// TwinCAT 3 PLC project PalettenstationPLC
// ProgramVersion: 3.1.4022.7
// libraries:
//   Tc2_Standard, * (Beckhoff Automation GmbH)
//   Tc2_System, * (Beckhoff Automation GmbH)
//   Tc3_Module, * (Beckhoff Automation GmbH)
// project tree:
//   GVLs/ GVL_IO.TcGVL, GVL_Simulation.TcGVL
//   / PlcTask.TcTTO
//   POUs/ MAIN.TcPOU, FB_NotHalt.TcPOU
//   DUTs/ E_StoppKategorie.TcDUT
// real-time tasks:
//   TASK PlcTask: cycle T#10ms, priority 20, ADS port 350
//   TASK Task_IO: cycle T#10ms, priority 1, ADS port 301
// I/O:
//   DEVICE Gerät 1 (EtherCAT), AmsNetId 5.35.203.54.2.1
//     Klemme 1 (EK1100) [EK1100 EtherCAT-Koppler (2A E-Bus)]
//       Klemme 2 (EL1002) [EL1002 2K. Dig. Eingang 24V, 3ms]
//       Klemme 3 (EL1004) [EL1004 4K. Dig. Eingang 24V, 3ms]
//       Klemme 4 (EL1004) [EL1004 4K. Dig. Eingang 24V, 3ms]
//       Klemme 5 (EL1008) [EL1008 8K. Dig. Eingang 24V, 3ms]
//       Klemme 6 (EL2004) [EL2004 4K. Dig. Ausgang 24V, 0.5A]
//       Klemme 7 (EL2004) [EL2004 4K. Dig. Ausgang 24V, 0.5A]
//       Klemme 8 (EL2008) [EL2008 8K. Dig. Ausgang 24V, 0.5A]
//       Klemme 9 (EL3064) [EL3064 4K.Ana. Eingang 0-10V]
//       Klemme 10 (EL3144) [EL3144 4K. Ana. Eingang 0-20mA]
//       Klemme 11 (EL3204) [EL3204 4K. Ana. Eingang PT100 (RTD)]
//       Klemme 12 (EL4014) [EL4014 4K. Ana. Ausgang 0-20mA, 12bit]
//       Klemme 13 (EL3681) [EL3681 Digitale Multimeter Klemme]
//       Klemme 14 (EK1110) [EK1110 EtherCAT-Verlängerung]

CONFIGURATION PalettenstationPLC
    RESOURCE PLC ON TwinCAT3
        TASK PlcTask(INTERVAL := T#10ms, PRIORITY := 20);
        PROGRAM MAIN WITH PlcTask : MAIN;
    END_RESOURCE
END_CONFIGURATION

// ---- DUTs/E_StoppKategorie.TcDUT
// =====================================================
// E_StoppKategorie
// =====================================================
// Bildet die Stoppkategorien nach EN 60204-1 als Software-Modell ab
// (siehe FB_NotHalt fuer den ausfuehrlichen Sicherheitshinweis).
// KEINE zertifizierte Sicherheitsklassifizierung.
// =====================================================
TYPE E_StoppKategorie :
(
	Kategorie_0 := 0,	// Sofortiger, unkontrollierter Halt durch Wegnahme der Energie/Freigabe
	Kategorie_1 := 1	// Kontrollierter Halt: Energie bleibt bis sicherer Zustand erhalten, danach Wegnahme
);
END_TYPE

// ---- GVLs/GVL_IO.TcGVL
{attribute 'qualified_only'}
VAR_GLOBAL

    // ==================================================
    // DIGITALE EINGÄNGE
    // ==================================================

    DI_NotHaltFrei        AT %I* : BOOL;
    DI_SchutzhaubeZu      AT %I* : BOOL;
    DI_PaletteEingang     AT %I* : BOOL;
    DI_PalettePositioniert AT %I* : BOOL;
    DI_HubUnten           AT %I* : BOOL;
    DI_HubOben            AT %I* : BOOL;
    DI_KollisionFrei      AT %I* : BOOL;
    DI_WerkerQuittierung  AT %I* : BOOL;


    // ==================================================
    // DIGITALE AUSGÄNGE
    // ==================================================

    DO_SignalGruen        AT %Q* : BOOL;
    DO_AlarmRot           AT %Q* : BOOL;
    DO_Foerderband        AT %Q* : BOOL;
    DO_FoerderbandStopp   AT %Q* : BOOL;
    DO_HubwerkHoch        AT %Q* : BOOL;
    DO_HubwerkRunter      AT %Q* : BOOL;
    DO_ProzessFreigabe    AT %Q* : BOOL;
    DO_Heizfreigabe       AT %Q* : BOOL;


    // ==================================================
    // ANALOGE EINGÄNGE
    // ==================================================

    AI_FolienTemperatur   AT %I* : REAL;
    AI_MotorTemperatur    AT %I* : REAL;

	// ==================================================
	// INTERNE PROGRAMMVARIABLEN
	// ==================================================

	Schritt : INT := 0;
	AlarmAktiv : BOOL := FALSE;

	// SIM_Aktiv = TRUE  -> Schrittkette nutzt GVL_Simulation-Werte
	// SIM_Aktiv = FALSE -> Schrittkette nutzt echte DI_*-Hardwareeingaenge (Default)
	SIM_Aktiv : BOOL := FALSE;


END_VAR

// ---- GVLs/GVL_Simulation.TcGVL
{attribute 'qualified_only'}
VAR_GLOBAL
	GVL_SIM_NotHaltFrei         : BOOL := TRUE;
    GVL_SIM_SchutzhaubeZu       : BOOL := TRUE;
    GVL_SIM_PaletteEingang      : BOOL := FALSE;
    GVL_SIM_PalettePositioniert : BOOL := FALSE;
    GVL_SIM_HubUnten            : BOOL := TRUE;
    GVL_SIM_HubOben             : BOOL := FALSE;
    GVL_SIM_KollisionFrei       : BOOL := TRUE;
    GVL_SIM_WerkerQuittierung   : BOOL := FALSE;
	GVL_SIM_FolienTemperatur  	: REAL := 175.0;
	GVL_SIM_MotorTemperatur   	: REAL := 50.0;
	
END_VAR

// ---- POUs/MAIN.TcPOU
PROGRAM MAIN
VAR
	tProzesszeit : TON;

	bNotHaltFrei         : BOOL;
    bSchutzhaubeZu       : BOOL;
    bPaletteEingang      : BOOL;
    bPalettePositioniert : BOOL;
    bHubUnten            : BOOL;
    bHubOben             : BOOL;
    bKollisionFrei       : BOOL;
    bWerkerQuittierung   : BOOL;

END_VAR

// =====================================================
// AUSGÄNGE ZU BEGINN JEDES SPS-ZYKLUS ZURÜCKSETZEN
// =====================================================

GVL_IO.DO_SignalGruen      := FALSE;
GVL_IO.DO_AlarmRot         := FALSE;
GVL_IO.DO_Foerderband      := FALSE;
GVL_IO.DO_FoerderbandStopp := FALSE;
GVL_IO.DO_HubwerkHoch      := FALSE;
GVL_IO.DO_HubwerkRunter    := FALSE;
GVL_IO.DO_ProzessFreigabe  := FALSE;
GVL_IO.DO_Heizfreigabe     := FALSE;


// =====================================================
// UMSCHALTUNG SIMULATION / HARDWARE
// =====================================================
// GVL_IO.SIM_Aktiv = TRUE  -> Werte aus GVL_Simulation
// GVL_IO.SIM_Aktiv = FALSE -> Werte von den echten %I*-Eingaengen (Default)

IF GVL_IO.SIM_Aktiv THEN

    bNotHaltFrei         := GVL_Simulation.GVL_SIM_NotHaltFrei;
    bSchutzhaubeZu       := GVL_Simulation.GVL_SIM_SchutzhaubeZu;
    bPaletteEingang      := GVL_Simulation.GVL_SIM_PaletteEingang;
    bPalettePositioniert := GVL_Simulation.GVL_SIM_PalettePositioniert;
    bHubUnten            := GVL_Simulation.GVL_SIM_HubUnten;
    bHubOben             := GVL_Simulation.GVL_SIM_HubOben;
    bKollisionFrei       := GVL_Simulation.GVL_SIM_KollisionFrei;
    bWerkerQuittierung   := GVL_Simulation.GVL_SIM_WerkerQuittierung;
	
    GVL_IO.AI_FolienTemperatur := GVL_Simulation.GVL_SIM_FolienTemperatur;
	GVL_IO.AI_MotorTemperatur  := GVL_Simulation.GVL_SIM_MotorTemperatur;
	
	

ELSE

    bNotHaltFrei         := GVL_IO.DI_NotHaltFrei;
    bSchutzhaubeZu       := GVL_IO.DI_SchutzhaubeZu;
    bPaletteEingang      := GVL_IO.DI_PaletteEingang;
    bPalettePositioniert := GVL_IO.DI_PalettePositioniert;
    bHubUnten            := GVL_IO.DI_HubUnten;
    bHubOben             := GVL_IO.DI_HubOben;
    bKollisionFrei       := GVL_IO.DI_KollisionFrei;
    bWerkerQuittierung   := GVL_IO.DI_WerkerQuittierung;

END_IF

// lesen -->  Programm ausführen -->  E/A schreiben --> wieder von vorne
// =====================================================
// SCHRITTKETTE
// =====================================================

CASE GVL_IO.Schritt OF

    0:// S0 - Anlage bereit und wartet auf Palette

        GVL_IO.DO_SignalGruen := TRUE;

        IF bNotHaltFrei
           AND bSchutzhaubeZu
           AND bHubUnten
           AND bPaletteEingang THEN

            GVL_IO.Schritt := 1;

        END_IF


    1: // S1 - Förderband transportiert Palette

        GVL_IO.DO_Foerderband := TRUE;

        IF NOT bNotHaltFrei THEN

            GVL_IO.Schritt := 8;

        ELSIF bPalettePositioniert THEN

            GVL_IO.Schritt := 2;

        END_IF


    2: // S2 - Palette stoppen

        GVL_IO.DO_FoerderbandStopp := TRUE;

        // Im nächsten SPS-Zyklus zu Hubwerk hoch
        GVL_IO.Schritt := 3;


    3: // S3 - Hubwerk fährt nach oben

        GVL_IO.DO_FoerderbandStopp := TRUE;
        GVL_IO.DO_HubwerkHoch      := TRUE;

        IF NOT bNotHaltFrei
           OR NOT bKollisionFrei THEN

            GVL_IO.Schritt := 8;

        ELSIF bHubOben THEN

            GVL_IO.Schritt := 4;

        END_IF


    4: // S4 - Temperatur prüfen

        GVL_IO.DO_FoerderbandStopp := TRUE;
        GVL_IO.DO_Heizfreigabe     := TRUE;

        IF GVL_IO.AI_MotorTemperatur > 100.0 THEN

            GVL_IO.Schritt := 8;

        ELSIF GVL_IO.AI_FolienTemperatur >= 165.0
           AND GVL_IO.AI_FolienTemperatur <= 185.0 THEN

            GVL_IO.Schritt := 5;

        ELSE

            GVL_IO.Schritt := 8;

        END_IF


    5: // S5 - Bearbeitung läuft fünf Sekunden

        GVL_IO.DO_FoerderbandStopp := TRUE;
        GVL_IO.DO_Heizfreigabe     := TRUE;
        GVL_IO.DO_ProzessFreigabe  := TRUE;

        tProzesszeit(
            IN := TRUE,
            PT := T#5S
        );

        IF GVL_IO.AI_FolienTemperatur < 165.0
           OR GVL_IO.AI_FolienTemperatur > 185.0
           OR GVL_IO.AI_MotorTemperatur > 100.0
           OR NOT bNotHaltFrei THEN

            tProzesszeit(IN := FALSE);
            GVL_IO.Schritt := 8;

        ELSIF tProzesszeit.Q THEN

            tProzesszeit(IN := FALSE);
            GVL_IO.Schritt := 6;

        END_IF


    6: // S6 - Hubwerk fährt nach unten

        GVL_IO.DO_FoerderbandStopp := TRUE;
        GVL_IO.DO_HubwerkRunter    := TRUE;

        IF NOT bNotHaltFrei THEN

            GVL_IO.Schritt := 8;

        ELSIF bHubUnten THEN

            GVL_IO.Schritt := 7;

        END_IF


    7: // S7 - Palette verlässt Station

        GVL_IO.DO_Foerderband := TRUE;

        IF NOT bPalettePositioniert THEN

            GVL_IO.Schritt := 0;

        END_IF


    8: // S8 - Alarm setzen

        GVL_IO.AlarmAktiv := TRUE;
        GVL_IO.Schritt := 9;


    9: // S9 - Warten auf Fehlerbeseitigung und Quittierung

        GVL_IO.DO_AlarmRot := TRUE;

        IF bWerkerQuittierung
           AND bNotHaltFrei
           AND GVL_IO.AI_FolienTemperatur >= 165.0
           AND GVL_IO.AI_FolienTemperatur <= 185.0
           AND GVL_IO.AI_MotorTemperatur <= 100.0 THEN

            GVL_IO.AlarmAktiv := FALSE;
            GVL_IO.Schritt := 0;

        END_IF


    ELSE // Unbekannter Schrittwert

        GVL_IO.AlarmAktiv := TRUE;
        GVL_IO.Schritt := 9;

END_CASE

END_PROGRAM

// ---- POUs/FB_NotHalt.TcPOU
// =====================================================
// FB_NotHalt - Software-Modell einer Not-Halt-Stoppkategorie
// =====================================================
// WICHTIGER HINWEIS (bitte nicht entfernen):
// Dies ist KEINE zertifizierte Sicherheitsfunktion nach EN ISO 13849-1 / IEC 62061.
// Der Baustein bildet nur das *Verhalten* der Stoppkategorien 0 und 1 nach
// EN 60204-1 in gewoehnlicher SPS-Logik nach - zu Lern- und Demonstrationszwecken
// in diesem Projekt (Standard-I/O, kein TwinCAT-Safety-System vorhanden).
//
// Fuer echte funktionale Sicherheit (Personenschutz) sind zwingend erforderlich:
//   - zertifizierte Safety-Hardware (z.B. TwinCAT Safety, EL69xx-Klemmen)
//   - zweikanalige/redundante Signalauswertung mit Querschlusserkennung
//   - Performance-Level-Nachweis nach EN ISO 13849-1 (bzw. SIL nach IEC 62061)
//   - ein durch die zustaendige Stelle abgenommenes Sicherheitskonzept
//
// Was dieser Baustein trotzdem zeigt:
//   - der Unterschied zwischen Kategorie 0 (sofortige Wegnahme der Energie)
//     und Kategorie 1 (kontrollierter Halt, dann Wegnahme) nach EN 60204-1
//   - Verriegelung (Latching) des Not-Halt-Zustands bis zu einer bewussten,
//     eigenstaendigen Wiederanlauf-Handlung (EN ISO 13850) - nicht identisch
//     mit einer allgemeinen Alarm-Quittierung
// =====================================================
FUNCTION_BLOCK FB_NotHalt
VAR_INPUT
	bNotHalt_Roh		: BOOL;				// Rohsignal Not-Halt-Taster (TRUE = ausgeloest)
	eKategorie			: E_StoppKategorie := E_StoppKategorie.Kategorie_0;
	bBewegungAktiv		: BOOL;				// Zusatzinfo fuer Kat.1: eine sicher zu beendende Bewegung laeuft noch
	bWiederanlaufTaste	: BOOL;				// separate, bewusste Wiederanlauf-Bestaetigung
	tMaxNachlauf		: TIME := T#2S;		// Obergrenze fuer den kontrollierten Nachlauf bei Kat.1
END_VAR
VAR_OUTPUT
	bFreigabeAntriebe	: BOOL;				// FALSE = alle Antriebe/Aktoren muessen sofort in den sicheren Zustand
	bVerriegelt			: BOOL;				// TRUE = Anlage bleibt gesperrt bis bewusster Wiederanlauf
	sZustand			: STRING(80);
END_VAR
VAR
	tNachlauf			: TON;
	bLatched			: BOOL;
END_VAR

IF bNotHalt_Roh THEN
	bLatched := TRUE;
END_IF

IF bLatched THEN

	CASE eKategorie OF

		E_StoppKategorie.Kategorie_0:
			// Kat. 0: sofortige, unkontrollierte Wegnahme der Freigabe
			bFreigabeAntriebe := FALSE;
			tNachlauf(IN := FALSE);
			sZustand := 'NOT-HALT Kat.0 - Antriebe sofort aus';

		E_StoppKategorie.Kategorie_1:
			// Kat. 1: Freigabe bleibt, bis der sichere Zustand erreicht ist,
			// danach Wegnahme - begrenzt auf eine maximale Nachlaufzeit.
			IF bBewegungAktiv THEN
				tNachlauf(IN := TRUE, PT := tMaxNachlauf);
				bFreigabeAntriebe := NOT tNachlauf.Q;
				sZustand := 'NOT-HALT Kat.1 - kontrollierter Nachlauf';
			ELSE
				tNachlauf(IN := FALSE);
				bFreigabeAntriebe := FALSE;
				sZustand := 'NOT-HALT Kat.1 - sicherer Zustand erreicht, Antriebe aus';
			END_IF

	ELSE
		// unbekannte Kategorie -> auf der sicheren Seite wie Kat. 0 behandeln
		bFreigabeAntriebe := FALSE;
		tNachlauf(IN := FALSE);
		sZustand := 'NOT-HALT - unbekannte Kategorie, sofortiger Halt';

	END_CASE

	bVerriegelt := TRUE;

	// Wiederanlauf erfordert eine EIGENSTAENDIGE, bewusste Aktion (EN ISO 13850) -
	// nicht identisch mit einer allgemeinen Alarm-Quittierung, und nur moeglich,
	// wenn die Rohausloesung selbst nicht mehr ansteht.
	IF NOT bNotHalt_Roh AND bWiederanlaufTaste THEN
		bLatched := FALSE;
		bVerriegelt := FALSE;
		tNachlauf(IN := FALSE);
		sZustand := 'Wiederanlauf bestaetigt - Anlage frei';
	END_IF

ELSE
	bFreigabeAntriebe := TRUE;
	bVerriegelt := FALSE;
	sZustand := 'Kein NOT-HALT aktiv';
END_IF

END_FUNCTION_BLOCK
